// TwinCAT 3 PLC project PLC_Project
// ProgramVersion: 3.1.4024.0
// libraries:
//   Tc2_Standard, * (Beckhoff Automation GmbH)
//   Tc2_System, * (Beckhoff Automation GmbH)
//   Tc3_Module, * (Beckhoff Automation GmbH)
//   VisuSymbols,3.5.10.0,System
// project tree:
//   / GlobalTextList.TcGTLO, PlcTask.TcTTO
//   POUs/ Control_Panel_Sequencer.TcPOU, FSM_States.TcDUT, MAIN.TcPOU
//   VISUs/ Sequencer_Visualization.TcVIS, VisualizationManager.TcVMO (not stored)
// real-time tasks:
//   TASK PlcTask: cycle T#10ms, priority 20, ADS port 350

CONFIGURATION PLC_Project
    RESOURCE PLC ON TwinCAT3
        TASK PlcTask(INTERVAL := T#10ms, PRIORITY := 20);
        PROGRAM MAIN WITH PlcTask : MAIN;
    END_RESOURCE
END_CONFIGURATION

// ---- POUs/FSM_States.TcDUT
{attribute 'qualified_only'}
{attribute 'strict'}
TYPE FSM_States :
(
	Startup_Idle 				:= 1,
	Startup_Power_Check 		:= 2,
	Startup_Breaker_Engage 		:= 3,
	Startup_Control_Power_On 	:= 4,
	Startup_Complete 			:= 5,
	Shutdown_Request 			:= 6,
	Fault_Present 				:= 8,
	Emergency_Stop 				:= 9
);
END_TYPE

// ---- POUs/MAIN.TcPOU
PROGRAM MAIN
VAR
END_VAR

Control_Panel_Sequencer();

END_PROGRAM

// ---- POUs/Control_Panel_Sequencer.TcPOU
PROGRAM Control_Panel_Sequencer
VAR
	State						:	INT				:=	FSM_States.Startup_Idle;
	
	MessageToOperator			:	STRING[255]		:=	'';
	CloseTimer					:	TON;
END_VAR

VAR_INPUT
	Control_Panel_Button_Start	:	BOOL			:=	FALSE;
	Control_Panel_Button_Stop	:	BOOL			:=	FALSE;
	Control_Panel_Button_E_Stop	:	BOOL			:=	FALSE;
	
	Voltage_Available			:	BOOL			:=	FALSE;
	Breaker_Closed_Feedback		:	BOOL			:=	FALSE;
END_VAR

VAR_OUTPUT
	Breaker_Close_Command		:	BOOL			:=	FALSE;
	Control_Circuits_Enable		:	BOOL			:=	FALSE;
	
	Status_Indication_On		:	BOOL			:=	FALSE;
	Status_Indication_Off		:	BOOL			:=	FALSE;
	Status_Indication_Fault		:	BOOL			:=	FALSE;
END_VAR

VAR CONSTANT
	CloseTime					:	TIME			:=	T#3S;
END_VAR

{Region "Sequencer"}
CASE State OF
	FSM_States.Startup_Idle:
		MessageToOperator		:=	'Conotrol Panel In Idle. Press Start Button To Continue';
		
		IF(Control_Panel_Button_Start)THEN
			State				:=	State + 1;
			MessageToOperator	:=	'Start Button Pressed';
		END_IF;
	FSM_States.Startup_Power_Check:
		IF(Voltage_Available)THEN
			State				:=	FSM_States.Startup_Breaker_Engage;
		ELSE
			State				:=	FSM_States.Fault_Present;
			MessageToOperator	:=	'No Voltage Is Present For Control Panel Operation';
		END_IF;
	FSM_States.Startup_Breaker_Engage:
		Breaker_Close_Command	:=	TRUE;
		
		//	Breaker Has XX Seconds In Which To Close Or Else A Fault May Be Present On The Device Or In The Circuit
		IF(NOT CloseTimer.Q)THEN
			CloseTimer(IN	:= 	TRUE,	PT	:=	CloseTime);
		ELSE
			CloseTimer(IN	:=	FALSE,	PT	:=	CloseTime);
			
			//	Check Breaker Feedback Matches Up With Breaker Command Signal
			IF(Breaker_Closed_Feedback)THEN
				State				:=	State + 1;
				MessageToOperator	:=	'Breaker Closed Successfully';
			ELSE
				State				:=	FSM_States.Fault_Present;
				MessageToOperator	:=	'Breaker Failed To Close';
			END_IF;		
		END_IF;
	FSM_States.Startup_Control_Power_On:
		Control_Circuits_Enable		:=	TRUE;
		MessageToOperator			:=	'Enabling Control Circuits';
		
		IF(NOT CloseTimer.Q)THEN
			CloseTimer(IN	:=	TRUE,	PT	:=	CloseTime);
		ELSE
			State					:=	State + 1;
			CloseTimer(IN	:=	FALSE,	PT	:=	CloseTime);
		END_IF;
	FSM_States.Startup_Complete:
			MessageToOperator		:=	'Startup Successfull! Panel Is Ready To Run';
			
			Status_Indication_On	:=	TRUE;
			Status_Indication_Off	:=	FALSE;
			Status_Indication_Fault	:=	FALSE;
			
			//	Check For Stop Command
			IF(Control_Panel_Button_Stop)THEN
				State				:=	State + 1;
			END_IF;
			
			//	Check For Emergency Stop Command
			IF(Control_Panel_Button_Stop)THEN
				State				:=	FSM_States.Emergency_Stop;
			END_IF;
	FSM_States.Shutdown_Request:
			State					:=	FSM_States.Startup_Idle;
			Control_Circuits_Enable	:=	FALSE;
			Breaker_Close_Command	:=	FALSE;
	FSM_States.Fault_Present:
			Status_Indication_Fault	:=	TRUE;
			MessageToOperator		:=	'Fault Detected';
	FSM_States.Emergency_Stop:
			Control_Circuits_Enable	:=	FALSE;
			Breaker_Close_Command	:=	FALSE;
			MessageToOperator		:=	'Emergency Stop Active';
	ELSE
		MessageToOperator			:=	'Unknown Sequence State Requested!';	
END_CASE;
{endregion}

END_PROGRAM

// ---- VISUs/Sequencer_Visualization.TcVIS
VISUALIZATION Sequencer_Visualization  // 2x2
END_VISUALIZATION
